PROGRAM Stn053_51_Stn221MainMergePrestop
VAR
//correct
	{attribute 'TcLinkToOSO' := '.iPuckPresent   :=  <0,1,2>TIIB[N48S00 (AL1332)]^N48S01 (AL2341)^TxPDO^input byte 0;
								 .iBufferFull   :=  <0,1,2>TIIB[N48S00 (AL1332)]^N48S01 (AL2341)^TxPDO^input byte 2;
								 .oStopLower   :=  <0,1,1>TIIB[N48S00 (AL1332)]^N48S02 (EX260)^RxPDO^output byte 0'}
	fbConvStop: FB_ConvStop;
END_VAR

//  This code instantiates a component that is implimented as a common function block
//    Note that I/O is linked directly to I/O variables inside the named instance

gStn053_51_Stn221MainMergePrestop.ConvRunning  := gConsumed_SafetyInterfaceConv.MtrRunning.Enc056Mtr08;

fbConvStop(
	pStn := ADR(gStn053),
	pCmp := ADR(gStn053_51_Stn221MainMergePrestop),
	pUpstreamStop := 0,
	pStateTraceBuffer := ADR(gStn053_StateTraceBuffer),
	pStateTraceFifo := ADR(gStn053_StateTraceFifo),
	pStats := ADR(gStn053_02_Stats));

END_PROGRAM

(* stored: Version 1.1.0.1, ProductVersion 3.1.4024.6
   POU Stn053_51_Stn221MainMergePrestop: Id {32331f4e-7500-44d1-8717-187fc8d17efb}, SpecialFunc None *)
